(* CoDeSys 2.3.9.62 project: Semaforo11_7.pro *)
(* Libraries: Standard.lib 2.6.14 10:37:46, IecSfc.lib 2.6.14 10:37:46 *)

(* Global variable list: Global_Variables *)
VAR_GLOBAL

 (* Entradas *)
	M: BOOL;

      (*Salidas*)
	Rojo: BOOL;    	(* Luz roja*)
	Amarillo:BOOL;	(* Luz amarilla *)
	Verde:BOOL;		(* Luz verde *)

      (* CONTADOR *)
      Conta:CTU;

END_VAR

(* POU PLC_PRG, LD *)
  PROGRAM PLC_PRG
VAR

	Eoff: BOOL;
	EV: BOOL;
	EA: BOOL;
	ER: BOOL;
	TempoVerde: TON;
	TempoAmarillo: TON;
	Flanco: R_TRIG;
	Aux: BOOL;
	TempoROjo: TON;
END_VAR
VAR (* helpers for the ST form of the networks *)
	_p1 : BOOL;
	_p2 : BOOL;
END_VAR
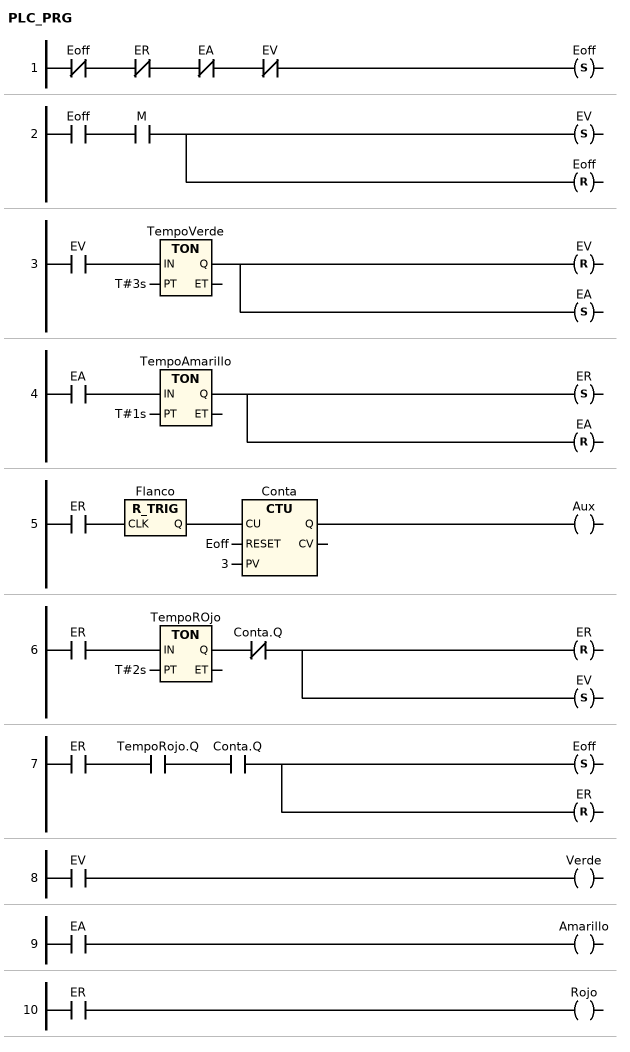
_LD_ (* Ladder Diagram *)
NETWORK 1
	[/Eoff] - [/ER] - [/EA] - [/EV] --- (S Eoff)
NETWORK 2
	[Eoff] - [M] --- (S EV) (R Eoff)
NETWORK 3
	[EV] - TempoVerde:TON(IN: *, PT: T#3s) --- (R EV) (S EA)
NETWORK 4
	[EA] - TempoAmarillo:TON(IN: *, PT: T#1s) --- (S ER) (R EA)
NETWORK 5
	[ER] - Flanco:R_TRIG(CLK: *) - Conta:CTU(CU: *, RESET: Eoff, PV: 3) --- (Aux)
NETWORK 6
	[ER] - TempoROjo:TON(IN: *, PT: T#2s) - [/Conta.Q] --- (R ER) (S EV)
NETWORK 7
	[ER] - [TempoRojo.Q] - [Conta.Q] --- (S Eoff) (R ER)
NETWORK 8
	[EV] --- (Verde)
NETWORK 9
	[EA] --- (Amarillo)
NETWORK 10
	[ER] --- (Rojo)
_END_LD_
(* the same logic as Structured Text *)
(* Network 1 *)
IF NOT Eoff AND NOT ER AND NOT EA AND NOT EV THEN Eoff := TRUE; END_IF;
(* Network 2 *)
_p1 := Eoff AND M;
IF _p1 THEN EV := TRUE; Eoff := FALSE; END_IF;
(* Network 3 *)
TempoVerde(IN := EV, PT := T#3s);
IF TempoVerde.Q THEN EV := FALSE; EA := TRUE; END_IF;
(* Network 4 *)
TempoAmarillo(IN := EA, PT := T#1s);
IF TempoAmarillo.Q THEN ER := TRUE; EA := FALSE; END_IF;
(* Network 5 *)
Flanco(CLK := ER);
Conta(CU := Flanco.Q, RESET := Eoff, PV := 3);
Aux := Conta.Q;
(* Network 6 *)
TempoROjo(IN := ER, PT := T#2s);
IF TempoROjo.Q AND NOT Conta.Q THEN ER := FALSE; EV := TRUE; END_IF;
(* Network 7 *)
_p2 := ER AND TempoRojo.Q AND Conta.Q;
IF _p2 THEN Eoff := TRUE; ER := FALSE; END_IF;
(* Network 8 *)
Verde := EV;
(* Network 9 *)
Amarillo := EA;
(* Network 10 *)
Rojo := ER;
END_PROGRAM

(* Visualisation SemaforoSimple
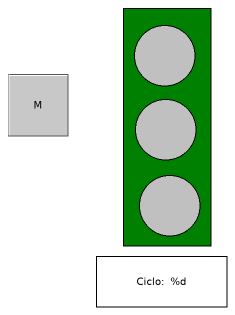
ellipse at (156,41)-(217,102): alarm colour if Rojo
ellipse at (157,115)-(218,176): alarm colour if Amarillo
ellipse at (161,191)-(222,252): alarm colour if Verde
rectangle at (118,272)-(249,323): text "Ciclo:  %d"; shows CONTA.CV
button at (30,90)-(90,152): text "M"; taps M
1 more shapes without text or variables
*)
